TYPE ST_LogMsg :
STRUCT
	DateandTime : STRING(24);
	Status : E_StatusCode; 
	StatusDescription : WSTRING;
	ItemID : DINT;
END_STRUCT
END_TYPE

(* stored: Version 1.1.0.1, ProductVersion 3.1.4024.4
   DUT ST_LogMsg: Id {df2f2379-ed09-4e8c-9735-3e258bc032ae} *)
